{attribute 'qualified_only'}
VAR_GLOBAL CONSTANT
	FurElise : ARRAY [0..100] OF  Mus_Sounds :=[
 	(note := E_Notes.NOTE_E5,              tempo:= 9),
                (note := E_Notes.NOTE_DS5,  tempo:=    9),
                (note := E_Notes.NOTE_E5,    tempo:=   9),
                (note := E_Notes.NOTE_DS5,   tempo:=   9),
                (note := E_Notes.NOTE_E5,    tempo:=   9),
                (note := E_Notes.NOTE_B4,    tempo:=   9),
                (note := E_Notes.NOTE_D5,    tempo:=   9),
                (note := E_Notes.NOTE_C5,    tempo:=   9),
                (note := E_Notes.NOTE_A4,    tempo:=   3),
                (note := E_Notes.NOTE_C4,    tempo:=   9),
                (note := E_Notes.NOTE_E4,    tempo:=   9),
                (note := E_Notes.NOTE_A4,    tempo:=   9),
                (note := E_Notes.NOTE_B4,     tempo:=  3),
                (note := E_Notes.NOTE_E4,    tempo:=   9),
                (note := E_Notes.NOTE_GS4,    tempo:=  9),
                (note := E_Notes.NOTE_B4,    tempo:=          9),
                (note := E_Notes.NOTE_C5,    tempo:=   3),
                (note := E_Notes.NOTE_E4,    tempo:=   9),
                (note := E_Notes.NOTE_E5,    tempo:=   9),
                (note := E_Notes.NOTE_DS5,   tempo:=   9),
                (note := E_Notes.NOTE_E5,    tempo:=   9),
                (note := E_Notes.NOTE_DS5,   tempo:=   9),
                (note := E_Notes.NOTE_E5,    tempo:=   9),
                (note := E_Notes.NOTE_B4,    tempo:=   9),
                (note := E_Notes.NOTE_D5,   tempo:=    9),
                (note := E_Notes.NOTE_C5,   tempo:=    9),
                (note := E_Notes.NOTE_A4,    tempo:=   3),
                (note := E_Notes.NOTE_C4,    tempo:=   9),
                (note := E_Notes.NOTE_E4,    tempo:=   9),
                (note := E_Notes.NOTE_A4,    tempo:=   9),
                (note := E_Notes.NOTE_B4,    tempo:=   3),
                (note := E_Notes.NOTE_E4,    tempo:=          9),
                (note := E_Notes.NOTE_C5,    tempo:=   9),
                (note := E_Notes.NOTE_B4,   tempo:=    9),
                (note := E_Notes.NOTE_A4,    tempo:=   3),
                (note := E_Notes.NOTE_B4,    tempo:=   9),
                (note := E_Notes.NOTE_C5,    tempo:=   9),
                (note := E_Notes.NOTE_D5,    tempo:=   9),
                (note := E_Notes.NOTE_E5,    tempo:=   3),
                (note := E_Notes.NOTE_G4,    tempo:=   9),
                (note := E_Notes.NOTE_F5,    tempo:=   9),
                (note := E_Notes.NOTE_E5,    tempo:=   9),
                (note := E_Notes.NOTE_D5,     tempo:=  3),
                (note := E_Notes.NOTE_F4,     tempo:=  9),
                (note := E_Notes.NOTE_E5,    tempo:=   9),
                (note := E_Notes.NOTE_D5,    tempo:=   9),
                (note := E_Notes.NOTE_C5,    tempo:=   3),
                (note := E_Notes.NOTE_E4,    tempo:=          9),
                (note := E_Notes.NOTE_D5,   tempo:=    9),
                (note := E_Notes.NOTE_C5,    tempo:=   9),
                (note := E_Notes.NOTE_B4,    tempo:=   9),
                (note := E_Notes.NOTE_E4,    tempo:=   9),
                (note := E_Notes.NOTE_E5,   tempo:=    9),
                (note := E_Notes.NOTE_E4,    tempo:=   9),
                (note := E_Notes.NOTE_E5,    tempo:=   9),
                (note := E_Notes.NOTE_E4,    tempo:=   9),
                (note := E_Notes.NOTE_E5,    tempo:=   9),
                (note := E_Notes.NOTE_E4,     tempo:=  9),
                (note := E_Notes.NOTE_E5,    tempo:=   9),
                (note := E_Notes.NOTE_DS4,    tempo:=  9),
                (note := E_Notes.NOTE_E5,    tempo:=   9),
                (note := E_Notes.NOTE_D4,     tempo:=  9),
                (note := E_Notes.NOTE_E5,     tempo:=  9),
                (note := E_Notes.NOTE_DS4,   tempo:=        9),
                (note := E_Notes.NOTE_E5,    tempo:=   9),
                (note := E_Notes.NOTE_B4,    tempo:=   9),
                (note := E_Notes.NOTE_D5,    tempo:=   9),
                (note := E_Notes.NOTE_C5,    tempo:=   9),
                (note := E_Notes.NOTE_A4,     tempo:=  3),
                (note := E_Notes.NOTE_C4,     tempo:=  9),
                (note := E_Notes.NOTE_E4,    tempo:=   9),
                (note := E_Notes.NOTE_A4,    tempo:=   9),
                (note := E_Notes.NOTE_B4,    tempo:=   3),
                (note := E_Notes.NOTE_E4,    tempo:=   9),
                (note := E_Notes.NOTE_GS4,   tempo:=   9),
                (note := E_Notes.NOTE_B4,     tempo:=  9),
                (note := E_Notes.NOTE_C5,     tempo:=  3),
                (note := E_Notes.NOTE_E4,     tempo:=  9),
                (note := E_Notes.NOTE_E5,     tempo:=  9),
                (note := E_Notes.NOTE_DS5,    tempo:=       9),
                (note := E_Notes.NOTE_E5,    tempo:=   9),
                (note := E_Notes.NOTE_DS5,    tempo:=  9),
                (note := E_Notes.NOTE_E5,     tempo:=  9),
                (note := E_Notes.NOTE_B4,     tempo:=  9),
                (note := E_Notes.NOTE_D5,     tempo:=  9),
                (note := E_Notes.NOTE_C5,     tempo:=  9),
                (note := E_Notes.NOTE_A4,    tempo:=   3),
                (note := E_Notes.NOTE_C4,    tempo:=   9),
                (note := E_Notes.NOTE_E4,    tempo:=   9),
                (note := E_Notes.NOTE_A4,    tempo:=   9),
                (note := E_Notes.NOTE_B4,    tempo:=   3),
                (note := E_Notes.NOTE_E4,    tempo:=   8),
                (note := E_Notes.NOTE_C5,    tempo:=   8),
                (note := E_Notes.NOTE_B4,    tempo:=   8),
                (note := E_Notes.NOTE_A4,    tempo:=   1),
                (note := E_Notes.STOP,       tempo:=   9)
];

END_VAR

(* stored: Version 1.1.0.1, ProductVersion 3.1.4024.6
   GVL FurElise: Id {68e82930-8b3f-4271-880e-3f08433025b8} *)
